% RSLogix 500 project I2P Hands On Test 1.RSS, saved by version 10.00.00.00 %
PROJECT "UNTITLED"    % processor: Bul.1763 MicroLogix 1100 Series B %

PROGRAM FILES
  LAD 2   5 rungs

DATA FILES
  O0 OUTPUT  4 elements
  I1 INPUT  6 elements
  S2 STATUS  66 elements
  B3 BINARY  1 elements
  T4 TIMER  1 elements
  C5 COUNTER  1 elements
  R6 CONTROL  1 elements
  N7 INTEGER  1 elements
  F8 FLOAT  1 elements

LADDER 2
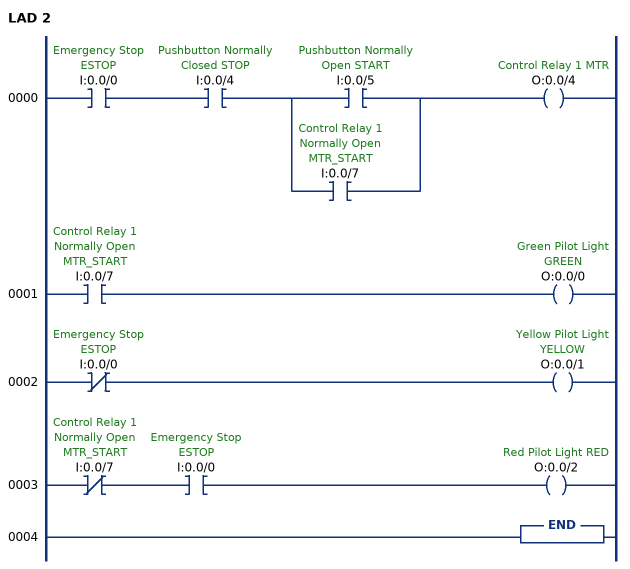
% Rung: 0 %
SOR XIC I:0.0/0 XIC I:0.0/4 BST XIC I:0.0/5 NXB XIC I:0.0/7 BND OTE O:0.0/4 EOR
%   I:0.0/0  ESTOP  "Emergency Stop" %
%   I:0.0/4  STOP  "Pushbutton Normally Closed" %
%   I:0.0/5  START  "Pushbutton Normally Open" %
%   I:0.0/7  MTR_START  "Control Relay 1 Normally Open" %
%   O:0.0/4  MTR  "Control Relay 1" %
% Rung: 1 %
SOR XIC I:0.0/7 OTE O:0.0/0 EOR
%   I:0.0/7  MTR_START  "Control Relay 1 Normally Open" %
%   O:0.0/0  GREEN  "Green Pilot Light" %
% Rung: 2 %
SOR XIO I:0.0/0 OTE O:0.0/1 EOR
%   I:0.0/0  ESTOP  "Emergency Stop" %
%   O:0.0/1  YELLOW  "Yellow Pilot Light" %
% Rung: 3 %
SOR XIO I:0.0/7 XIC I:0.0/0 OTE O:0.0/2 EOR
%   I:0.0/7  MTR_START  "Control Relay 1 Normally Open" %
%   I:0.0/0  ESTOP  "Emergency Stop" %
%   O:0.0/2  RED  "Red Pilot Light" %
% Rung: 4 %
SOR END EOR

OTHER DOCUMENTED ADDRESSES
  I:0.0/1  3PSSA  "3 Position Selector Switch Position A"
  I:0.0/2  3PSSB  "3 Position Selector Switch Position B"
  I:0.0/3  2PSS  "2 Position Selector Switch"
  I:0.0/6  PB3NO  "Pushbutton Normally Open"
  I:0.0/8  CR2NO  "Control Relay 2 Normally Open"
  I:0.0/9  REVMSNO  "Reverse Mtr. Starter Normally Open"
  O:0.0/3  BLUE  "Blue Pilot Light"
  O:0.0/5  CR2  "Control Relay 2"
